PROGRAM pouMsgS4
VAR
	
	
	
END_VAR

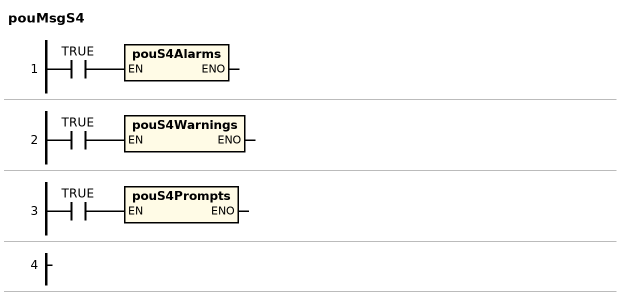
// NETWORK 1
pouS4Alarms();

// NETWORK 2
pouS4Warnings();

// NETWORK 3
pouS4Prompts();

// NETWORK 4

END_PROGRAM

(* stored: Version 1.1.0.1, ProductVersion 3.1.4024.12
   POU pouMsgS4: Id {1b8dd0fc-ce59-43eb-8f24-9efd796b1e82}, SpecialFunc None *)
